PROGRAM MAIN
VAR
	TON_UP: TON;
	TON_DOWN: TON;
	HalfCycle: TIME := T#50MS;
	FB_Blinker_0: FB_Blinker;


	bInifeBeat: BOOL;
	NT_StartProcess_HMI: NT_StartProcess;
	SR_StartProcess: SR;
	R_TRIG_0: R_TRIG;
	TON_StartProcess: TON;
END_VAR

LifeBeat();
//T_200ms := NOT T_200ms;

Carriage_Manager();
Turret_Manager();
CrossCut_Manager();
XDrive_Manager();
ZAxis_Manager();
KrAxis();
PRG_IO();

PRG_00_General();
PRG_01_Reel();
PRG_02_Xdrive();
	PRG_02_Xdrive.ACT_02_1_Xdrive();
PRG_03_Saw();
PRG_04_Turret();
	PRG_04_Turret.ACT_04_1_Turret();
PRG_05_Carriage();
	PRG_05_Carriage.ACT_05_1_Carriage();
PRG_06_CrossCut();
	PRG_06_CrossCut.ACT_06_1_CrossCut();
	PRG_06_CrossCut.ACT_06_2_CrossCutSpeed();
PRG_07_ZAxis();
	PRG_07_ZAxis.ACT_07_1_ZAxis();
PRG_08_AutoCrossCut();
	PRG_08_AutoCrossCut.ACT_08_1_AutoCrossCut();
PRG_09_HomePosition();
	PRG_09_HomePosition.ACT_09_HomePosition();
PRG_10_CrossCutPosition();
	PRG_10_CrossCutPosition.ACT_10_CrossCutPosition();
PRG_11_ScreenButtons();
PRG_12_ProductionReport();
PRG_90_GeneralConditions();
PRG_91_TwinSAFE();
PRG_99_Persistent();

ACTION LifeBeat:
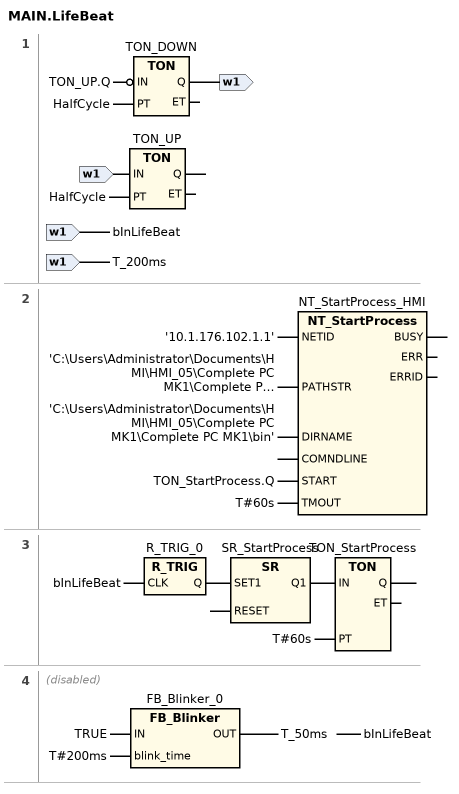
// NETWORK 1
TON_DOWN(IN := NOT TON_UP.Q, PT := HalfCycle); // TON
TON_UP(IN := TON_DOWN.Q, PT := HalfCycle); // TON
bInLifeBeat := TON_DOWN.Q;
T_200ms := TON_DOWN.Q;

// NETWORK 2
NT_StartProcess_HMI(
    NETID := '10.1.176.102.1.1',
    PATHSTR := 'C:\Users\Administrator\Documents\HMI\HMI_05\Complete PC MK1\Complete PC MK1\bin\ProgressControl.exe',
    DIRNAME := 'C:\Users\Administrator\Documents\HMI\HMI_05\Complete PC MK1\Complete PC MK1\bin',
    START := TON_StartProcess.Q,
    TMOUT := T#60s); // NT_StartProcess

// NETWORK 3
R_TRIG_0(CLK := bInLifeBeat); // R_TRIG
SR_StartProcess(SET1 := R_TRIG_0.Q); // SR
TON_StartProcess(IN := SR_StartProcess.Q1, PT := T#60s); // TON

// NETWORK 4 (disabled)
// FB_Blinker_0(IN := TRUE, blink_time := T#200ms); // FB_Blinker
// T_50ms := FB_Blinker_0.OUT;
// bInLifeBeat := FB_Blinker_0.OUT;
END_ACTION

END_PROGRAM

(* stored: Version 1.1.0.1, ProductVersion 3.1.4024.15
   POU MAIN: Id {802b1616-ec6a-40b9-9874-ea9048ad0dda}, SpecialFunc None
   Action LifeBeat: Id {83e498b2-7847-4ce9-95b4-c99e760d3c4a} *)
